RoboDK station: KUKAKR60_301119.rdk

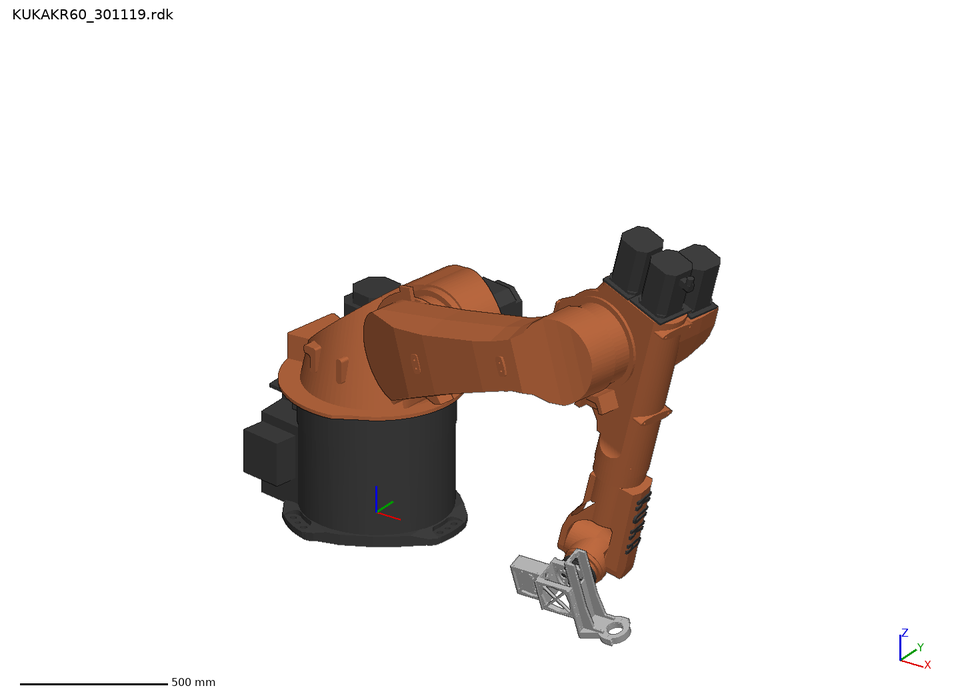
[picture v0: the station drawn from its stored meshes, robots at their saved joint values, targets as dots, program paths as lines]
Station KUKAKR60_301119. Poses are relative to the parent item; angles as X-Y-Z fixed-axis rotations.
  - frame KUKA KR 60 HA Base at (0, 0, 0) mm
    - robot KUKA KR 60 HA: 6 axes, payload 30 kg, reach 2033 mm, repeatability 0.05 mm, weight 665 kg
        modified DH rows (alpha deg, a mm, theta deg, d mm): 0, 0, 0, 815; -90, 350, 0, 0; 0, 850, -90, 0; -90, 145, 0, 820; 90, 0, 0, 0; -90, 0, 180, 170
        joint limits [-185, -135, -120, -350, -119, -350] to [185, 35, 158, 350, 119, 350]; home [0, -90, 90, 0, 0, 0]; saved at [9.93, -17.63, 123.642, 105.12, 73.498, -106.462]
      - tool ToolsHolder, TCP at (-150, 193, 118) mm, rotated rx 0 ry 0 rz 90 deg, size 419.4 x 326 x 130 mm
